FUNCTION_BLOCK AlarmEventLogger IMPLEMENTS Alarm
VAR
	alarm : FB_TcAlarm;
	_Source : Name;
	autoReset : BOOL;
END_VAR

PROPERTY Arguments : I_TcArguments
GET
Arguments := alarm.ipArguments;
END_GET
END_PROPERTY

METHOD Clear
VAR_INPUT
END_VAR
alarm.Clear(0, TRUE);
END_METHOD

METHOD ClearArguments : I_TcArguments
alarm.ipArguments.Clear();

IF (_Source <> 0) THEN
	alarm.ipArguments.AddStringByValue(value := _Source.Name);
END_IF

ClearArguments := alarm.ipArguments;
END_METHOD

METHOD FB_init : BOOL
VAR_INPUT
	bInitRetains : BOOL; // if TRUE, the retain variables are initialized (warm start / cold start)
	bInCopyCode : BOOL;  // if TRUE, the instance afterwards gets moved into the copy code (online change)
	
	event : TcEventEntry;
	autoReset : BOOL;
END_VAR
THIS^.autoReset := autoReset;
alarm.CreateEx(stEventEntry := event, bWithConfirmation := NOT autoReset, ipSourceInfo := 0);
END_METHOD

{attribute 'monitoring' := 'call'}
PROPERTY IsRaised : BOOL
GET
IsRaised := alarm.bRaised;
END_GET
END_PROPERTY

METHOD Raise
VAR_INPUT
END_VAR
IF (alarm.ipArguments.nCount = 0 AND _Source <> 0) THEN
	alarm.ipArguments.AddStringByValue(value := _Source.Name);
END_IF

alarm.Raise(0);
END_METHOD

{attribute 'monitoring' := 'call'}
PROPERTY Source : Name
GET
Source := _Source;
END_GET
SET
_Source := Source;
END_SET
END_PROPERTY

METHOD Watch
VAR_INPUT
	eventCondition : BOOL;
END_VAR
IF (eventCondition) THEN
	Raise();
ELSIF (autoReset AND IsRaised) THEN
	Clear();
END_IF
END_METHOD

END_FUNCTION_BLOCK

(* stored: Version 1.1.0.1
   POU AlarmEventLogger: Id {d0e3ccbe-965e-0019-3a52-a4d182233dd4}, SpecialFunc None
   Property Arguments: Id {345ff380-780b-0dd1-3ebd-e0daa03e2ebb}
   Get Get: Id {2a83c0c1-beb4-08e0-09dd-d2694feb9e33}
   Method Clear: Id {5e6685b2-9d9d-0bd6-0b80-36d17ef6c63d}
   Method ClearArguments: Id {a2932eac-18c7-04df-2451-3e41b4c10e96}
   Method FB_init: Id {13b93e8d-5b11-0a43-3eea-01e38a3c84d4}
   Property IsRaised: Id {cc265ab0-9ea0-0c78-2a6a-eea337dd7b8f}
   Get Get: Id {fb9a8cac-efab-0b9f-2a41-b0daa8278494}
   Method Raise: Id {96cfa2a4-23c7-0ebe-0c1d-3f6a3f94f801}
   Property Source: Id {9d3b7778-12fd-08b4-0b66-8744cc82ee16}
   Get Get: Id {9b6cbf4e-d561-0beb-307f-4e7d663fcad4}
   Set Set: Id {519a888e-b735-039a-24b9-068740b93537}
   Method Watch: Id {41dfdb64-d522-0299-0c10-fdb0f1d05e9f} *)
